TYPE TRunCmdReject :
	(
		RCR_None,
		RCR_OpenDrawer,
		RCR_LockDrawer,
		RCR_UnlockDrawer
	);
END_TYPE

(* stored: Version 1.1.0.1, ProductVersion 3.1.4022.12
   DUT TRunCmdReject: Id {b28b2bda-05bc-4e98-94b6-3d8a5c5a4945} *)
